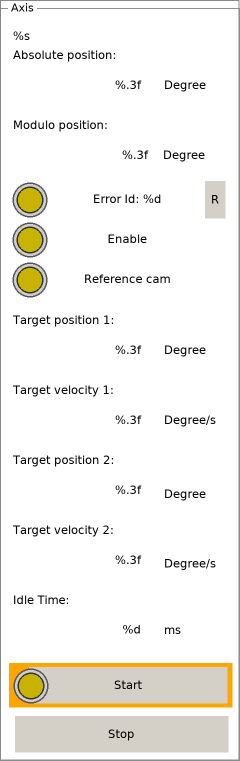
VISUALIZATION TplAxisReversingSequence  // 240x761
VAR_IN_OUT
	sAxisDescription				:STRING;
	fAbsolutePositon				:LREAL;
	fModuloPositon					:LREAL;
	bError							:BOOL;
	nErrorId						:DWORD;
	bReset							:BOOL;
	bPowerStatus					:BOOL;
	bReferenceCam					:BOOL;
	bRevSeqStart					:BOOL;
	bRevSeqStop						:BOOL;
	fRevSeqTargetPos1				:LREAL;
	fRevSeqTargetVelo1				:LREAL;
	fRevSeqTargetPos2				:LREAL;
	fRevSeqTargetVelo2				:LREAL;
	nRevSeqIdleTime					:UINT;
	bRevSeqDone						:BOOL;
	bRevSeqBusy						:BOOL;
END_VAR
    GroupBox (0,0 240x761), "Axis"
        Group (10,40 227x60)
            Rectangle (0,30 148x30), "%.3f", text variable: fAbsolutePositon
            Label (151,30 76x30), "Degree"
            Label (0,0 216x30), "Absolute position:"
        Group (10,180 200x40)
            Rectangle (20,1 195x36), "Error Id: %d", text variable: nErrorId
            Lamp1 (0,0 40x40), variable: bError, style: Lamp-Lamp1-Yellow
        Group (10,220 215x40)
            Rectangle (20,1 195x36), "Enable"
            Lamp1 (0,0 40x40), variable: bPowerStatus, style: Lamp-Lamp1-Yellow
        Group (10,260 215x40)
            Rectangle (20,1 195x36), "Reference cam"
            Lamp1 (0,0 40x40), variable: bReferenceCam, style: Lamp-Lamp1-Yellow
        Rectangle (205,181 20x37), "R", tooltip "Reset", colour toggle: bReset
            tap bReset
        Rectangle (10,25 230x22), "%s", text variable: sAxisDescription
        Rectangle (10,335 148x30), "%.3f", text variable: fRevSeqTargetPos1
            OnMouseClick: write the text variable via VisuDialogs.Numpad
        Label (161,335 76x30), "Degree"
        Label (10,305 216x30), "Target position 1:"
        Rectangle (10,405 148x30), "%.3f", text variable: fRevSeqTargetVelo1
            OnMouseClick: write the text variable via VisuDialogs.Numpad
        Label (161,405 76x30), "Degree/s"
        Group (10,110 230x60)
            Rectangle (0,30 148x30), "%.3f", text variable: fModuloPositon
            Label (150,30 80x30), "Degree"
            Label (0,0 200x30), "Modulo position:"
        Rectangle (9,663 223x44), invisible if: NOT bRevSeqBusy
        Rectangle (29,667 198x36), "Start", colour toggle: bRevSeqStart
            toggle bRevSeqStart
        Lamp1 (11,666 40x40), variable: bRevSeqDone, style: Lamp-Lamp1-Yellow
        Rectangle (15,716 213x36), "Stop", colour toggle: bRevSeqStop
            toggle bRevSeqStop
        Rectangle (10,615 148x29), "%d", text variable: nRevSeqIdleTime
            OnMouseClick: write the text variable via VisuDialogs.Numpad
        Label (10,585 216x30), "Idle Time:"
        Label (10,375 216x30), "Target velocity 1:"
    Label (161,479 76x30), "Degree"
    Rectangle (10,475 148x30), "%.3f", text variable: fRevSeqTargetPos2
        OnMouseClick: write the text variable via VisuDialogs.Numpad
    Label (10,445 216x30), "Target position 2:"
    Rectangle (10,545 148x30), "%.3f", text variable: fRevSeqTargetVelo2
        OnMouseClick: write the text variable via VisuDialogs.Numpad
    Label (161,549 76x29), "Degree/s"
    Label (10,515 216x30), "Target velocity 2:"
    Label (161,615 76x30), "ms"
END_VISUALIZATION

(* stored: Version 1.1.0.1
   Visu TplAxisReversingSequence: Id {d07d3152-58f8-4d11-a0e1-01f0624149a7} *)
